// TIA Portal V18 export
// export: Created 2026-06-08T17:01:58.2141032Z, ExportSetting WithDefaults, DisplayName Totally Integrated Automation Portal, DisplayVersion V18, DisplayName TIA Portal Openness, DisplayVersion V18, DisplayName TIA Portal Version Control Interface, DisplayVersion V18, DisplayName STEP 7 Professional, DisplayVersion V18, DisplayName STEP 7 Safety, DisplayVersion V18, DisplayName WinCC Professional, DisplayVersion V18
FUNCTION "MAIN_WIND_DOWN" : Void   // FC2, LAD
{ S7_Optimized_Access := 'TRUE' }
VERSION : 0.1
// stored: AutoNumber true, IsIECCheckEnabled false, SetENOAutomatically false, UDAEnableTagReadback false
BEGIN

REGION Network 1
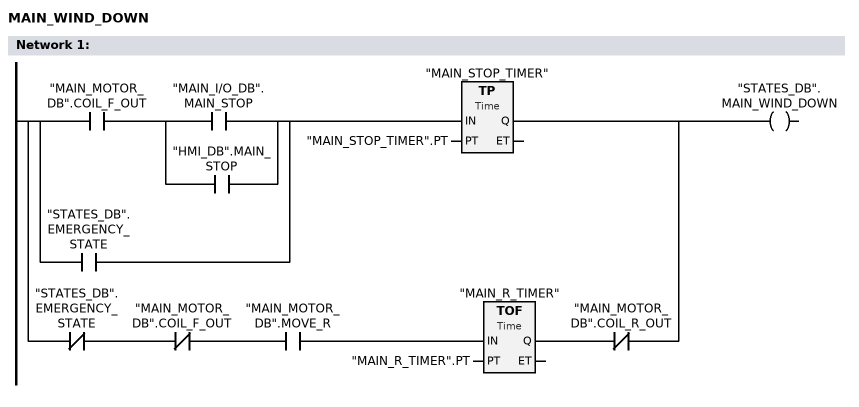
   RUNG wire#powerrail
      Contact( "MAIN_MOTOR_DB".COIL_F_OUT )
      wire#w1
      Contact( "MAIN_I/O_DB".MAIN_STOP )
      wire#w2
      { S7_Templates := "time_type := Time" } "MAIN_STOP_TIMER".TP(pt := "MAIN_STOP_TIMER".PT, et =>)
      wire#w3
      Coil( "STATES_DB".MAIN_WIND_DOWN )
   END_RUNG
   RUNG wire#w1
      Contact( "HMI_DB".MAIN_STOP )
   END_RUNG wire#w2
   RUNG wire#powerrail
      Contact( "STATES_DB".EMERGENCY_STATE )
   END_RUNG wire#w2
   RUNG wire#powerrail
      I_Contact( "STATES_DB".EMERGENCY_STATE )
      I_Contact( "MAIN_MOTOR_DB".COIL_F_OUT )
      Contact( "MAIN_MOTOR_DB".MOVE_R )
      { S7_Templates := "time_type := Time" } "MAIN_R_TIMER".TOF(pt := "MAIN_R_TIMER".PT, et =>)
      I_Contact( "MAIN_MOTOR_DB".COIL_R_OUT )
   END_RUNG wire#w3
   // the same network as SCL:
   "MAIN_STOP_TIMER".TP(IN := ("MAIN_MOTOR_DB".COIL_F_OUT AND ("MAIN_I/O_DB".MAIN_STOP OR "HMI_DB".MAIN_STOP)) OR "STATES_DB".EMERGENCY_STATE,
                        PT := "MAIN_STOP_TIMER".PT);
   "MAIN_R_TIMER".TOF(IN := NOT "STATES_DB".EMERGENCY_STATE AND NOT "MAIN_MOTOR_DB".COIL_F_OUT AND "MAIN_MOTOR_DB".MOVE_R,
                      PT := "MAIN_R_TIMER".PT);
   "STATES_DB".MAIN_WIND_DOWN := "MAIN_STOP_TIMER".Q OR ("MAIN_R_TIMER".Q AND NOT "MAIN_MOTOR_DB".COIL_R_OUT);
END_REGION
END_FUNCTION
